TYPE ACRMemoryByteEvents :
STRUCT
	_Values : ARRAY [0..GCL.cMemoryEventsMAX] OF ACRMemoryByteEvent;
END_STRUCT
END_TYPE

(* stored: Version 1.1.0.1, ProductVersion 3.1.4020.12
   DUT ACRMemoryByteEvents: Id {3c604f96-0b1b-4ec6-b9b2-d580cdb14528} *)
